FUNCTION_BLOCK CorrecionCaudalxOffset
VAR_INPUT
	Caudalimetro_inf	:REAL;
	Caudalimetro_sup	:REAL;	
	Inyeccion			:BOOL;
	Offset				:REAL;
END_VAR
VAR_OUTPUT
	PV					:REAL;
END_VAR
VAR
END_VAR

IF Not Inyeccion THEN
	PV:=Caudalimetro_sup*(Offset+1);
ELSE
	PV:=Caudalimetro_inf*(Offset+1);
END_IF

END_FUNCTION_BLOCK

(* stored: Version 1.1.0.1, ProductVersion 3.1.4024.12
   POU CorrecionCaudalxOffset: Id {090d73de-50aa-4d6d-85ee-0e5126d9f268}, SpecialFunc None *)
